FUNCTION_BLOCK FB_Event
VAR_INPUT
	nID:			INT;
	ipArguments:	Tc3_EventLogger.I_TcArguments;
END_VAR
VAR_OUTPUT
END_VAR
VAR
	sText:			STRING(255);
	sSeverity:		STRING;
	
	bInit:			BOOL := TRUE;
	bIsRaised:		BOOL;
	
	
	fbArguments:	FB_Arguments;
END_VAR

ipArguments := fbArguments;

IF			bInit THEN
	bInit := FALSE;
	fbArguments.sOriginalString := sText;
END_IF

fbArguments(sOutText => sText, iInterfacePointer := ipArguments);

PROPERTY bRaised : Bool
GET
bRaised := bIsRaised;
END_GET
END_PROPERTY

METHOD Clear
VAR_INPUT
	a:	INT;
	b: BOOL;

END_VAR
bIsRaised := FALSE;
EventLogger.unpinEvent(nID);
END_METHOD

METHOD Raise
VAR_INPUT
	a:	INT;
END_VAR
bIsRaised := TRUE;
sText := fbArguments.sOutText;
EventLogger.logEvent(nID, sText,sSeverity, TRUE);
END_METHOD

METHOD RequestEventText
VAR_INPUT
	a:	INT;
END_VAR
VAR_IN_OUT
	b:	STRING(255);
END_VAR
VAR_INPUT
	c:	INT;
END_VAR
b := sText;
END_METHOD

METHOD send
VAR_INPUT
	a:	INT;
END_VAR
sText := fbArguments.sOutText;
EventLogger.logEvent(nID, sText,sSeverity, FALSE);
END_METHOD

METHOD setText
VAR_INPUT
	sSeverity:			STRING;
	sText:				STRING(255);
END_VAR
THIS^.sSeverity := sSeverity;
THIS^.sText := sText;
END_METHOD

END_FUNCTION_BLOCK

(* stored: Version 1.1.0.1, ProductVersion 3.1.4024.12
   POU FB_Event: Id {89a7a39d-d29e-4485-8727-034be5441a2a}, SpecialFunc None
   Property bRaised: Id {cd918912-3ed8-4b97-b728-92a6a1a90877}
   Get Get: Id {c515fc13-ddf1-470d-9fdc-e7e061add2b5}
   Method Clear: Id {49a59f45-c26f-480e-a5e8-140695b0c0e0}
   Method Raise: Id {4120ae0f-71dc-4e79-9ed1-627f83fbcb3e}
   Method RequestEventText: Id {1d294914-c055-42f6-b179-a221e4bc3b4c}
   Method send: Id {84687f39-e6e2-43e1-aa05-d87252ebd670}
   Method setText: Id {613ec003-d685-425a-9b1b-efa397c63bac} *)
